TYPE "SpeedMachine_DataOut"
VERSION : 0.1
// Block: SpeedMachine_DataOut
   STRUCT
      Fan_M_Contactor : Bool;
   END_STRUCT;

END_TYPE
